// TwinCAT 3 PLC project state_machine_prj
// ProgramVersion: 3.1.4024.0
// libraries:
//   Tc2_Standard, * (Beckhoff Automation GmbH)
//   Tc2_System, * (Beckhoff Automation GmbH)
//   Tc2_Utilities, * (Beckhoff Automation GmbH)
//   Tc3_Module, * (Beckhoff Automation GmbH)
//   VisuDialogs, * (System)
// project tree:
//   DUTs/ ST_MyData.TcDUT
//   / GlobalTextList.TcGTLO, PlcTask.TcTTO, Visualization Manager.TcVMO (not stored)
//   POUs/ Class Diagram.TcCD (not stored), FB_ChargedState.TcPOU, FB_DischargeState.TcPOU, FB_DisconnectedState.TcPOU, FB_ErrorState.TcPOU, FB_FileWriter.TcPOU, FB_IdleState.TcPOU, FB_MACHINE.TcPOU, FB_PrechargeState.TcPOU, I_State.TcIO, MAIN.TcPOU
//   VISUs/ Visualisation.TcVIS
// (motion and I/O tree: see PLC project safety)
// real-time tasks:
//   TASK Safety: cycle T#5ms, priority 6, ADS port 350
//   TASK StateMachine: cycle T#1ms, priority 4, ADS port 351
// variable links:
//   safety/safety Instance <-> state_machine_prj/state_machine_prj Instance
//     PlcTask Outputs/MAIN.b_ESTOPout <-> PlcTask Inputs/MAIN.b_estop
//     PlcTask Outputs/MAIN.b_LED <-> PlcTask Inputs/MAIN.b_resetLed
//     PlcTask Outputs/MAIN.b_SafetyStateOut <-> PlcTask Inputs/MAIN.b_reset
//   state_machine_prj/state_machine_prj Instance <-> Device 5 (EtherCAT)/Term 1 (EK1100)/Term 2 (EL3702)
//     PlcTask Inputs/MAIN.n_A_sensors[0] <-> Ch2 Sample 0/Ch2 Value
//     PlcTask Inputs/MAIN.n_A_sensors[1] <-> Ch1 Sample 0/Ch1 Value
//   state_machine_prj/state_machine_prj Instance <-> Device 5 (EtherCAT)/Term 1 (EK1100)/Term 4 (EL3702)
//     PlcTask Inputs/MAIN.n_V_sensors[0] <-> Ch1 Sample 0/Ch1 Value
//     PlcTask Inputs/MAIN.n_V_sensors[1] <-> Ch2 Sample 0/Ch2 Value
//   state_machine_prj/state_machine_prj Instance <-> Device 5 (EtherCAT)/Term 1 (EK1100)/Term 6 (EL1004)
//     PlcTask Inputs/MAIN.b_bypass_contactors_fb[0] <-> Channel 3/Input
//     PlcTask Inputs/MAIN.b_bypass_contactors_fb[1] <-> Channel 4/Input
//     PlcTask Inputs/MAIN.b_main_contactors_fb[0] <-> Channel 1/Input
//     PlcTask Inputs/MAIN.b_main_contactors_fb[1] <-> Channel 2/Input
//   state_machine_prj/state_machine_prj Instance <-> Device 5 (EtherCAT)/Term 1 (EK1100)/Term 7 (EL2004)
//     PlcTask Outputs/MAIN.b_bypass_contactors[0] <-> Channel 3/Output
//     PlcTask Outputs/MAIN.b_bypass_contactors[1] <-> Channel 4/Output
//     PlcTask Outputs/MAIN.b_main_contactors[0] <-> Channel 1/Output
//     PlcTask Outputs/MAIN.b_main_contactors[1] <-> Channel 2/Output

CONFIGURATION state_machine_prj
    RESOURCE PLC ON TwinCAT3
        TASK PlcTask(INTERVAL := T#1ms, PRIORITY := 4);
        PROGRAM MAIN WITH PlcTask : MAIN;
    END_RESOURCE
END_CONFIGURATION

// ---- DUTs/ST_MyData.TcDUT
TYPE ST_MyData :
STRUCT
    Id          : UDINT;
    Value       : REAL;
    Timestamp   : T_MaxString; 
END_STRUCT
END_TYPE

// ---- POUs/I_State.TcIO
INTERFACE I_State

METHOD PUBLIC Check
END_METHOD

PROPERTY PUBLIC Description : STRING
GET
END_GET
END_PROPERTY

METHOD PUBLIC PressButton
END_METHOD

METHOD PUBLIC PressDischarge
END_METHOD

METHOD PUBLIC Reset
END_METHOD

METHOD PUBLIC Stop
END_METHOD

METHOD PUBLIC TimerDone
END_METHOD

END_INTERFACE

// ---- POUs/MAIN.TcPOU
PROGRAM MAIN
// Variables, constants ... are created (instanced) here
VAR
	(* Inputs *)
	n_V_sensors 				AT %I* 		: ARRAY[0..1] OF INT; // defining 2 elements array of INT type as input to the PLC task
	n_A_sensors 				AT %I*		: ARRAY[0..1] OF INT; 
	
	b_reset						AT %I*		: BOOL;
	b_estop						AT %I*		: BOOL;

	b_main_contactors_fb 		AT %I* 		: ARRAY[0..1] OF BOOL; // defining 4 elements array of BOOL type as input of feedback for the contactors to the PLC task
	b_bypass_contactors_fb 		AT %I* 		: ARRAY[0..1] OF BOOL;
	
	b_resetLed					AT %I*		: BOOL; 
	
	(* Outputs *)
	b_main_contactors			AT %Q*		: ARRAY[0..1] OF BOOL; // defining 4 elements array of BOOL type as outpout to the PLC task
	b_bypass_contactors			AT %Q*		: ARRAY[0..1] OF BOOL;

	(* FB_MACHINE *) 
	b_user_button							: BOOL := FALSE;
	b_discharge								: BOOL := FALSE;
	n_lower_boundV							: INT := 380;
	n_upper_boundV							: INT := 460; 
	n_minV 									: INT := 5;
	
	t_max_time								: TIME := T#250MS; //5x the time constant for a RC circuit with R=100ohms and C=235µF
	
	fbMachine 								: FB_MACHINE(nLowerBoundV := n_lower_boundV,
													     nUpperBoundV := n_upper_boundV,
													     nMinV := n_minV,
													     tMaxTime := t_max_time); 
	(*Visualisation variables*)
    sState         							: STRING;
	n_V_sensors_scaled 						: ARRAY[0..1] OF REAL; // defining 2 elements array of INT type as input to the PLC task
	n_A_sensors_scaled						: ARRAY[0..1] OF REAL;
	sLog									: ARRAY[0..19] OF STRING(600); 
	
	(* FILE_WRITER VARIABLES *) 
	sFilePath 								: STRING := 'C:\Users\Administrator\Desktop\AXav-Precharge_Curbs\'; //default file path for the data
    
	arrVoltageData    						: ARRAY [0..1] OF ST_MyData;
	arrCurrentData							: ARRAY [0..1] OF ST_MyData;
	arrBypassData							: ARRAY [0..1] OF ST_MyData;
	arrMainData								: ARRAY [0..1] OF ST_MyData;
	
    nIteration      						: UDINT:=0;
    bStartNewJob    						: BOOL := FALSE; // When set to false the FileWriter is active
	bFirstLoop								: BOOL := TRUE; // Allows to write the header of the file on the first loop (then it will be set to FALSE for the rest of the task)
	tStartTime								: TIME;
	
	fbVoltage1								: FB_FileWriter; 
	fbCurrent1								: FB_FileWriter; 
	fbVoltage2								: FB_FileWriter;
	fbCurrent2								: FB_FileWriter;
	fbBypass1								: FB_FileWriter;
	fbBypass2								: FB_FileWriter; 
	fbMain1									: FB_FileWriter; 
	fbMain2									: FB_FileWriter; 
	
	fbFormatString  						: FB_FormatString;
	fbFormatString1  						: FB_FormatString;
	fbFormatString2							: FB_FormatString; 
	fbFormatString3							: FB_FormatString;
	
	sHeader									: STRING := 'ID;VALUE;TIMESTAMP$n';

	n_Idx									: INT := 0;
	fileBlocks 								: ARRAY[0..3] OF  FB_FileWriter := [fbCurrent1, fbCurrent2, fbVoltage1, fbVoltage2];
	fileBlocksContactors					: ARRAY[0..3] OF  FB_FileWriter := [fbBypass1, fbBypass2, fbMain1, fbMain2];
    s_fileNames 							: ARRAY[0..3] OF STRING := ['SupplyCurrent.txt', 'LoadCurrent.txt', 'SupplyVoltage.txt', 'LoadVoltage.txt'];
	s_fileNamesContactors					: ARRAY[0..3] OF STRING := ['BypassContactor1.txt', 'BypassContactor2.txt', 'MainContactor1.txt', 'MainContactor2.txt'];
	s_FBStates								: ARRAY[0..3] OF STRING;
	s_FBStatesContactors					: ARRAY[0..3] OF STRING; 
END_VAR

(* ---------------------------- STATE MACHINE ------------------------------- *) 
fbMachine.Run(
			bAck:=b_user_button, 
			bDischarge := b_discharge, 
			nVSensors := n_V_Sensors, 
			nASensors := n_A_Sensors, 
			bBypassContactorsFB := b_bypass_contactors_fb,
			bMainContactorsFB := b_main_contactors_fb,
			bReset := b_reset,
			bESTOP := b_estop,
			bMainContactors => b_main_contactors, 
			bBypassContactors => b_bypass_contactors,
			);

(* --------------------- Visualisation properties ---------------------- *) 
// I need to link local variables with "fbMachine" properties because it is not possible to link a visualisation object (e.g. textbox) with a function box property
sState := fbMachine.ipState.Description;
n_V_sensors_scaled := fbMachine.VSensors; 
n_A_sensors_scaled := fbMachine.ASensors; 
sLog := fbMachine.Logs; 

(* --------------------- Data Saving ----------------------------- *)	
FOR n_Idx := 0 TO 3 DO
	fileBlocks[n_Idx](
		sFileName := s_fileNames[n_Idx],
		sFilePath := sFilePath,
		sNetId    := '');
		
	fileBlocksContactors[n_Idx](
		sFileName := s_fileNamesContactors[n_Idx],
		sFilePath := sFilePath,
		sNetId    := '');
			
	s_FBStates[n_Idx] := fileBlocks[n_Idx].FileWriteState; // STRING states to display in the visualisation file
	s_FBStatesContactors[n_Idx] := fileBlocksContactors[n_Idx].FileWriteState; // STRING states to display in the visualisation file
END_FOR	

IF bFirstLoop THEN // On the first loop
	FOR n_Idx := 0 TO 3 DO
		fileBlocks[n_Idx].WriteToFile(message := sHeader); // write the header of the file 
		fileBlocksContactors[n_Idx].WriteToFile(message := sHeader); // write the header of the file 
	END_FOR	
	tStartTime := TIME();
	bFirstLoop := FALSE;
END_IF

IF bStartNewJob THEN 
	// save the new data to the struct variable
	FOR n_Idx := 0 TO 1 DO
		arrVoltageData[n_Idx].Id := nIteration;
		arrVoltageData[n_Idx].Value := n_V_sensors_scaled[n_Idx];
		arrVoltageData[n_Idx].Timestamp := DINT_TO_STRING(TO_DINT(TIME() - tStartTime));
	
		arrCurrentData[n_Idx].Id := nIteration;
		arrCurrentData[n_Idx].Value :=n_A_sensors_scaled[n_Idx];
		arrCurrentData[n_Idx].Timestamp := DINT_TO_STRING(TO_DINT(TIME() - tStartTime)); 
		
		arrBypassData[n_Idx].Id := nIteration;
		arrBypassData[n_Idx].Value := BOOL_TO_REAL(b_bypass_contactors_fb[n_Idx]);
		arrBypassData[n_Idx].Timestamp := DINT_TO_STRING(TO_DINT(TIME() - tStartTime));
	
		arrMainData[n_Idx].Id := nIteration;
		arrMainData[n_Idx].Value :=BOOL_TO_REAL(b_main_contactors[n_Idx]);
		arrMainData[n_Idx].Timestamp := DINT_TO_STRING(TO_DINT(TIME() - tStartTime)); 
	END_FOR
	// write the data in the text file 
	FOR n_Idx := 0 TO 1 DO
		fbFormatString(
			sFormat := '%d;%f;%s$n',
			arg1    := F_UDINT(arrCurrentData[n_Idx].Id),
			arg2    := F_REAL(arrCurrentData[n_Idx].Value),
			arg3    := F_STRING(arrCurrentData[n_Idx].Timestamp));
		fileBlocks[n_Idx].WriteToFile(fbFormatString.sOut);
		fbFormatString1(
			sFormat := '%d;%f;%s$n',
			arg1    := F_UDINT(arrVoltageData[n_Idx].Id),
			arg2    := F_REAL(arrVoltageData[n_Idx].Value),
			arg3    := F_STRING(arrVoltageData[n_Idx].Timestamp));
		fileBlocks[n_Idx+2].WriteToFile(fbFormatString1.sOut);
		fbFormatString2(
			sFormat := '%d;%f;%s$n',
			arg1    := F_UDINT(arrBypassData[n_Idx].Id),
			arg2    := F_REAL(arrBypassData[n_Idx].Value),
			arg3    := F_STRING(arrBypassData[n_Idx].Timestamp));
		fileBlocksContactors[n_Idx].WriteToFile(fbFormatString2.sOut);
		fbFormatString3(
			sFormat := '%d;%f;%s$n',
			arg1    := F_UDINT(arrMainData[n_Idx].Id),
			arg2    := F_REAL(arrMainData[n_Idx].Value),
			arg3    := F_STRING(arrMainData[n_Idx].Timestamp));
		fileBlocksContactors[n_Idx+2].WriteToFile(fbFormatString3.sOut);
	END_FOR
	nIteration := nIteration + 1;
END_IF

END_PROGRAM

// ---- POUs/FB_MACHINE.TcPOU
FUNCTION_BLOCK PUBLIC FB_MACHINE

VAR_INPUT
	nVSensors 		 				: ARRAY[0..1] OF INT; // 2 INT elements array which contains the voltage sensors outputs
	nASensors 						: ARRAY[0..1] OF INT; // 2 INT elements array whihch contains the current sensors outputs
	
	(* Pre-Charge Timer *) 
	tMaxTime						: TIME; // Maximum pre-charge time
	
	(* Voltage boundaries *) 
	nLowerBoundV					: INT; // Input voltage lower bound (~50V) 
	nUpperBoundV					: INT; // Input voltage upper bound (~200V)
	nMinV							: INT; // Minimum voltage to leave "disconnected" state
	
	(* Timer *)
	charge_TON						: TON; 
END_VAR

VAR_OUTPUT
	ipState 						: I_State := fbDisconnectedState; // Current State of the state machine (default is FB_DisconnectedState)
END_VAR

VAR (* Internal variables *)
	fbDisconnectedState 			: FB_DisconnectedState(THIS);	
	fbIdleState 					: FB_IdleState(THIS); 
	fbPrechargeState 				: FB_PrechargeState(THIS); 
	fbChargedState					: FB_ChargedState(THIS); 
	fbDischargeState				: FB_DischargeState(THIS);
	fbErrorState					: FB_ErrorState(THIS);
	
	(* Sensors scaling *) 
	n_idx_1 						: INT := 0; 
	fVSensorsScaled 				: ARRAY[0..1] OF REAL; // defining 2 elements array of REAL type as internal variables
	fASensorsScaled 				: ARRAY[0..1] OF REAL; 
	
	(* Message log *) 
	sLog 							: ARRAY [0..19] OF STRING(600);
	nCount							: UINT := 0; // Keeps track of the number of elements in the array	
	nArraySize 						: UINT := 20; // Edit value if size of sLog changes 
	tLaunchTime 					: TIME; 	
	sMessage						: STRING(600);
	sPrevMessage					: STRING(600);
	
	(* Contactors *)
	bMainContactors					: ARRAY[0..1] OF BOOL; 
	bBypassContactors 				: ARRAY[0..1] OF BOOL; 
	
	(* Contactors feedback *)
	bMainContactorsFB				: ARRAY[0..1] OF BOOL; // defining 2 elements array of BOOL type as input of feedback for the main contactors to the PLC task
	bBypassContactorsFB				: ARRAY[0..1] OF BOOL; // defining 2 elements array of BOOL type as input of feedback for the precharge contactors to the PLC task

	(* Triggers *) 
	rtrigButtonAck					: R_TRIG; // Define trigger for user button 
	rtrigButtonDisch				: R_TRIG; 
	
	(* Misc *) 
	nRunCounter						: UINT := 10;
END_VAR

tLaunchTime := TIME(); // Reference point for log messages

METHOD PRIVATE AddToLog
VAR_INPUT
	sMsgINPUT			: STRING(600); //different from Message that doesn't contain the time tag
END_VAR
VAR
	nIdx 				: UINT := 0;
END_VAR
// IF the ARRAY is full, remove the first element 
IF NOT(Message = PrevMessage) THEN // NOT sMsgINPUT BECAUSE IT CONTAINS THE TIME TAG which will make it always different from PrevMessage
	IF THIS^.nCount = THIS^.nArraySize THEN
		FOR nIdx := 0 TO THIS^.nArraySize - 2 DO 
			sLog[nIdx] := sLog[nIdx + 1 ]; // shift the whole array
		END_FOR
		sLog[THIS^.nCount - 1] := sMsgINPUT; // Add the new string as the last elemnt of the array
	ELSE
		sLog[THIS^.nCount] := sMsgINPUT;
		THIS^.nCount := THIS^.nCount + 1;
	END_IF 
	THIS^.PrevMessage := Message;
END_IF
END_METHOD

PROPERTY PUBLIC ASensors : ARRAY[0..1] OF REAL
GET
ASensors := THIS^.fASensorsScaled;
END_GET
END_PROPERTY

PROPERTY PUBLIC BypassContactors : ARRAY[0..1] OF BOOL
GET
BypassContactors := THIS^.bBypassContactors;
END_GET
SET
THIS^.bBypassContactors := BypassContactors;
END_SET
END_PROPERTY

PROPERTY PRIVATE BypassContactorsFB : ARRAY[0..1] OF BOOL
GET
BypassContactorsFB := THIS^.bBypassContactorsFB;
END_GET
SET
THIS^.bBypassContactorsFB := BypassContactorsFB;
END_SET
END_PROPERTY

PROPERTY PUBLIC ChargedState : I_State
GET
ChargedState := THIS^.fbChargedState;
END_GET
END_PROPERTY

METHOD CheckContactors
VAR
	nIdx							: INT := 0; 
	
	bMainContactorsCheck 			: BOOL := TRUE; // true means that there is no problem
	bBypassContactorsCheck 			: BOOL := TRUE; 
	bConclusion 					: BOOL := TRUE; // true means that there is no problem
	
	fbDischargeState				: FB_DischargeState(THIS);
END_VAR
FOR nIdx := 0 TO 1 DO 
	bMainContactorsCheck := THIS^.bMainContactors[nIdx] = THIS^.bMainContactorsFB[nIdx]; // checks that the feedback signal corresponds to the contactor state
	bBypassContactorsCheck := THIS^.bBypassContactors[nIdx] = THIS^.bBypassContactorsFB[nIdx];
	
	IF NOT(bMainContactorsCheck) THEN
		THIS^.Message := CONCAT('[CheckContactors] The ', CONCAT(INT_TO_STRING(nIdx), ' Main contactor state does not match the signal sent'));
		bConclusion := FALSE; 
	END_IF
	IF NOT(bBypassContactorsCheck) THEN
		THIS^.Message := CONCAT('[CheckContactors] The ', CONCAT(INT_TO_STRING(nIdx), ' Bypass contactor state does not match the signal sent'));
		bConclusion := FALSE; 
	END_IF
END_FOR 

IF NOT(bConclusion) THEN
	THIS^.Message := CONCAT(THIS^.Message, '[CheckContactors]$A0 THE SYSTEM IS NOW BEING DISHCARGED');  
	THIS^.SetState(fbDischargeState);
	bConclusion := TRUE;
END_IF
END_METHOD

PROPERTY PUBLIC DischargeState : I_State
GET
DischargeState :=  THIS^.fbDischargeState;
END_GET
END_PROPERTY

PROPERTY PUBLIC DisconnectedState : I_State
GET
DisconnectedState := THIS^.fbDisconnectedState;
END_GET
END_PROPERTY

PROPERTY PUBLIC ErrorState : I_State
GET
ErrorState := THIS^.fbErrorState;
END_GET
END_PROPERTY

METHOD FB_init 
VAR_INPUT
	bInitRetains : BOOL; // if TRUE, the retain variables are initialized (warm start / cold start)
	bInCopyCode : BOOL;  // if TRUE, the instance afterwards gets moved into the copy code (online change)
	
	(* Pre-Charge Timer *) 
	tMaxTime						: TIME; 
	
	(* Voltage boundaries *) 
	nLowerBoundV					: INT; // Input voltage lower bound (~50V) 
	nUpperBoundV					: INT; // Input voltage upper bound (~200V)
	nMinV							: INT; // Minimum voltage to leave "disconnected" state
END_VAR
THIS^.tMaxTime := tMaxTime;
THIS^.nLowerBoundV := nLowerBoundV; 
THIS^.nUpperBoundV := nUpperBoundV; 
THIS^.nMinV := nMinV;
END_METHOD

PROPERTY PUBLIC IdleState : I_State
GET
IdleState := THIS^.fbIdleState;
END_GET
END_PROPERTY

PROPERTY PUBLIC Logs : ARRAY[0..19] OF STRING(600)
GET
Logs := THIS^.sLog;
END_GET
END_PROPERTY

PROPERTY PUBLIC LowerBoundV : INT
GET
LowerBoundV := THIS^.nLowerBoundV;
END_GET
SET
THIS^.nLowerBoundV := LowerBoundV;
END_SET
END_PROPERTY

PROPERTY PUBLIC MainContactors : ARRAY[0..1] OF BOOL
GET
MainContactors := THIS^.bMainContactors;
END_GET
SET
THIS^.bMainContactors := MainContactors;
END_SET
END_PROPERTY

PROPERTY PRIVATE MainContactorsFB : ARRAY[0..1] OF BOOL
GET
MainContactorsFB := THIS^.bMainContactorsFB;
END_GET
SET
THIS^.bMainContactorsFB := MainContactorsFB;
END_SET
END_PROPERTY

PROPERTY PUBLIC Message : STRING(600)
GET // PUBLIC
Message := THIS^.sMessage;
END_GET
SET // PUBLIC
THIS^.sMessage := Message; 
// Adds the difference between the laucnh time and the current time at the beginning of the log message
THIS^.AddToLog(CONCAT(CONCAT(CONCAT('[', TIME_TO_STRING(TIME()-THIS^.tLaunchTime)), '] '), THIS^.sMessage));
END_SET
END_PROPERTY

PROPERTY PUBLIC MinV : INT
GET
MinV := THIS^.nMinV;
END_GET
SET
THIS^.nMinV := MinV;
END_SET
END_PROPERTY

PROPERTY PUBLIC PrechargeState : I_State
GET
PrechargeState := THIS^.fbPrechargeState;
END_GET
END_PROPERTY

PROPERTY PrevMessage : STRING(600)
GET
PrevMessage := THIS^.sPrevMessage;
END_GET
SET
THIS^.sPrevMessage := PrevMessage;
END_SET
END_PROPERTY

METHOD PUBLIC Run
VAR_INPUT
	(* User buttons *)
	bAck							: BOOL; // User "next state" button
	bDischarge						: BOOL; // User "discharge" trigger button
	
	(* Sensors *)
	nVSensors 		 				: ARRAY[0..1] OF INT; // defining 2 elements array of INT type as input to the PLC task
	nASensors 						: ARRAY[0..1] OF INT; 
	
	bMainContactorsFB				: ARRAY[0..1] OF BOOL; 
	bBypassContactorsFB				: ARRAY[0..1] OF BOOL;
	
	bReset							: BOOL; // Reset signal
	bESTOP							: BOOL; // TRUE when the button is pressed
END_VAR

VAR
END_VAR

VAR_OUTPUT
	bMainContactors					: ARRAY[0..1] OF BOOL; 
	bBypassContactors				: ARRAY[0..1] OF BOOL;
END_VAR
(* ------------------------------------- SAFETY ------------------------------------ *)
//E-Stop check
IF NOT(bESTOP) THEN	
	ipState.Stop(); // sets state to ErrorState
	ipState.Check(); 
	bMainContactors := THIS^.MainContactors; 
	bBypassContactors := THIS^.BypassContactors;
	RETURN;
END_IF
//Reset check
IF ipState = ErrorState AND bReset THEN // reset has been pressed 
	ipState.Reset();
END_IF
// Functionning contactors check
IF RunCounter MOD 15 = 0  THEN // Checks contactors every 15 run loop because it takes some time for the feedback to adjust
	CheckContactors(); // Ensures that the contactors signals are the same as the contactors states
END_IF


(* ---------------------------------- STATE MACHINE ------------------------------------ *) 

(*Contactors*)
THIS^.MainContactorsFB := bMainContactorsFB;
THIS^.BypassContactorsFB := bBypassContactorsFB;

(* Buttons*) 
rtrigButtonAck(CLK := bAck); // Sets trigger for bUserButton variable 
rtrigButtonDisch(CLK := bDischarge); 

(*Sensors*)
THIS^.nVSensors := nVSensors;
THIS^.nASensors := nASensors; 

(* Timer configuration *) 
charge_TON(PT := THIS^.tMaxTime);

THIS^.ScaleSensors(); // Scaling the values of the sensors which will be used in the state machine 

IF (charge_TON.Q) THEN
	ipState.TimerDone(); // Used for the precharge state 
END_IF

IF (rtrigButtonDisch.Q) THEN
	ipState.PressDischarge();
END_IF

IF (rtrigButtonAck.Q) THEN
	ipState.PressButton();
END_IF

ipState.Check(); 

// Output of the state machine
bMainContactors := THIS^.MainContactors; 
bBypassContactors := THIS^.BypassContactors;
RETURN;
END_METHOD

PROPERTY PRIVATE RunCounter : UINT
GET
RunCounter := THIS^.nRunCounter;
END_GET
SET
THIS^.nRunCounter := RunCounter;
END_SET
END_PROPERTY

METHOD PRIVATE ScaleSensors
// Scaling of V sensors
FOR n_idx_1 := 0 TO 1 DO
	fVSensorsScaled[n_idx_1] := 1000*INT_TO_REAL(THIS^.nVSensors[n_idx_1])/32768;
	// e.g., if 1000 V on sensor --> card measures +10V --> software value = 32767 --> scaling is therefore 1000*VAL/32768
END_FOR

FOR n_idx_1 := 0 TO 1 DO
	fASensorsScaled[n_idx_1] := 25*INT_TO_REAL(THIS^.nASensors[n_idx_1])/32768; 
END_FOR
END_METHOD

METHOD INTERNAL SetState
VAR_INPUT
	newState		: I_State;
END_VAR
THIS^.ipState := newState;
END_METHOD

PROPERTY PUBLIC UpperBoundV : INT
GET
UpperBoundV := THIS^.nUpperBoundV;
END_GET
SET
THIS^.nUpperBoundV := UpperBoundV;
END_SET
END_PROPERTY

PROPERTY PUBLIC VSensors : ARRAY[0..1] OF REAL
GET
VSensors := THIS^.fVSensorsScaled;
END_GET
END_PROPERTY

END_FUNCTION_BLOCK

// ---- POUs/FB_DisconnectedState.TcPOU
FUNCTION_BLOCK INTERNAL FB_DisconnectedState IMPLEMENTS I_State
VAR
	pMachine		: POINTER TO FB_Machine; // Points to the state machine (THIS)
	fVSensors		: ARRAY[0..1] OF REAL; 
END_VAR

METHOD PUBLIC Check
VAR
	fInputVoltage 		: REAL; 
END_VAR
THIS^.ResetContactors(); //THE CONTACTORS NEED TO ALWAYS BE OPEN IN THIS STATE
fVSensors := THIS^.pMachine^.VSensors;
fInputVoltage := fVSensors[0];

IF (fInputVoltage >= THIS^.pMachine^.MinV) THEN
	THIS^.pMachine^.Message := '[DISCONNECTED] The input voltage is >= than the minimum voltage. $0A WAITING FOR ACKNOWLEDGEMENT TO ENTER IDLE STATE;';
ELSE 
	THIS^.pMachine^.Message := '[DISCONNECTED]The input voltage is <= than the minimum voltage.';
END_IF
END_METHOD

PROPERTY PUBLIC Description : STRING
GET
Description := 'DISCONNECTED';
END_GET
END_PROPERTY

METHOD PUBLIC FB_init
VAR_INPUT
	bInitRetains 	: BOOL; // if TRUE, the retain variables are initialized (warm start / cold start)
	bInCopyCode 	: BOOL;  // if TRUE, the instance afterwards gets moved into the copy code (online change)
	pMachine		: POINTER TO FB_Machine; // Points to the state machine (THIS)
END_VAR
THIS^.pMachine := pMachine;
END_METHOD

METHOD PUBLIC PressButton 
VAR
	//fbIdleSTate		: FB_IdleState(THIS^.pMachine); => variable for changing state method that causes a PLC bug
	fInputVoltage		: REAL; 
END_VAR
fVSensors := THIS^.pMachine^.VSensors;
fInputVoltage := fVSensors[0];

IF (fInputVoltage >= THIS^.pMachine^.MinV) THEN
		//THIS^.pMachine^.SetState(fbIdleState); => changing state method that causes a PLC bug
		THIS^.pMachine^.Message := '[DISCONNECTED] Acknowledge button has been pressed. $0A SYSTEM ENTERS IDLE STATE.';
		THIS^.pMachine^.SetState(THIS^.pMachine^.IdleState);
END_IF
END_METHOD

METHOD PUBLIC PressDischarge
END_METHOD

METHOD PUBLIC Reset
END_METHOD

METHOD PUBLIC ResetContactors
VAR
	nIdx					: INT := 0; 
	bBypassContactors		: ARRAY[0..1] OF BOOL; 
	bMainContactors			: ARRAY[0..1] OF BOOL; 
END_VAR
FOR nIdx := 0 TO 1 BY 1 DO 
	bBypassContactors[nIdx] := FALSE;
	bMainContactors[nIdx] := FALSE; 
END_FOR

THIS^.pMachine^.BypassContactors := bBypassContactors; // Reset every contactor 
THIS^.pMachine^.MainContactors := bMainContactors;
END_METHOD

METHOD PUBLIC Stop
THIS^.pMachine^.SetState(THIS^.pMachine^.ErrorState);
END_METHOD

METHOD PUBLIC TimerDone
END_METHOD

END_FUNCTION_BLOCK

// ---- POUs/FB_IdleState.TcPOU
FUNCTION_BLOCK INTERNAL FB_IdleState IMPLEMENTS I_State
VAR
	pMachine				: POINTER TO FB_Machine; // Points to the state machine (THIS)
	fVSensors				: ARRAY [0..1] OF REAL; 
END_VAR

METHOD PUBLIC Check 
VAR
	fInputVoltage			: REAL;	
END_VAR
fVSensors := THIS^.pMachine^.VSensors;

fInputVoltage := fVSensors[0];

IF (fInputVoltage >= THIS^.pMachine^.LowerBoundV AND fInputVoltage <= THIS^.pMachine^.UpperBoundV) THEN
	THIS^.pMachine^.Message := '[IDLE]The input voltage is within the boundaries.$0A NOW WAITING FOR ACKNOWLEDGEMENT TO ENTER PRE-CHARGE STATE.';
ELSE
	THIS^.pMachine^.Message := '[IDLE] The input voltage is NOT within the boundaries.$0A SYSTEM ENTERS DISCHARGE STATE.';
	THIS^.pMachine^.SetState(THIS^.pMachine^.DischargeState);
END_IF
END_METHOD

PROPERTY PUBLIC Description : STRING
GET
Description := 'IDLE';
END_GET
END_PROPERTY

METHOD PUBLIC FB_init
VAR_INPUT
	bInitRetains 	: BOOL; // if TRUE, the retain variables are initialized (warm start / cold start)
	bInCopyCode 	: BOOL;  // if TRUE, the instance afterwards gets moved into the copy code (online change)
	pMachine		: POINTER TO FB_Machine; // Points to the state machine (THIS)
END_VAR
THIS^.pMachine := pMachine;
END_METHOD

METHOD PUBLIC PressButton
VAR
	fInputVoltage			: REAL; 
END_VAR
fVSensors := THIS^.pMachine^.VSensors;
fInputVoltage := fVSensors[0];

IF (fInputVoltage >= THIS^.pMachine^.LowerBoundV AND fInputVoltage <= THIS^.pMachine^.UpperBoundV) THEN
	THIS^.pMachine^.Message := '[IDLE] Acknowledge button has been pressed. $0A SYSTEM ENTERS PRECHARGE STATE.';
	THIS^.pMachine^.SetState(THIS^.pMachine^.PrechargeState);
	THIS^.StartTimer();
END_IF
END_METHOD

METHOD PUBLIC PressDischarge
THIS^.pMachine^.Message := '[IDLE] Discharge button has been pressed. $0A SYSTEM ENTERS DISCHARGE STATE.';
THIS^.pMachine^.SetState(THIS^.pMachine^.DischargeState);
END_METHOD

METHOD PUBLIC Reset
THIS^.pMachine^.Message := '[IDLE] Reset button has been pressed. $0A SYSTEM ENTERS DISCHARGE STATE.';
THIS^.pMachine^.SetState(THIS^.pMachine^.DischargeState);
END_METHOD

METHOD PUBLIC StartTimer
THIS^.pMachine^.charge_TON.IN := TRUE; // Starts the Timer
END_METHOD

METHOD PUBLIC Stop
THIS^.pMachine^.SetState(THIS^.pMachine^.ErrorState);
END_METHOD

METHOD PUBLIC TimerDone
END_METHOD

END_FUNCTION_BLOCK

// ---- POUs/FB_PrechargeState.TcPOU
FUNCTION_BLOCK INTERNAL FB_PrechargeState  IMPLEMENTS I_State
VAR
	pMachine				: POINTER TO FB_Machine; // Points to the state machine (THIS)
	fVSensors				: ARRAY [0..1] OF REAL;
END_VAR

METHOD PUBLIC Check
VAR
	fLoadVoltage			: REAL;
	fInputVoltage 			: REAL;
END_VAR
THIS^.SetMainContactors();
fVSensors := THIS^.pMachine^.VSensors;

fInputVoltage := fVSensors[0];
fLoadVoltage := fVSensors[1];

IF (fLoadVoltage > 1.1 * fInputVoltage) THEN
	(* If the load voltage is greater than 110% of the input voltage then we consider that there is a problem and the load is disconnected *)
	THIS^.pMachine^.Message := '[PRECHARGE] The load voltage is greater than 110 percent of the input voltage.$0A THE SYSTEM ENTERS DISCHARGE STATE';
	THIS^.pMachine^.SetState(THIS^.pMachine^.DischargeState); 
	
ELSIF (fLoadVoltage <= 1.1 * fInputVoltage AND fLoadVoltage >= 0.9502 * fInputVoltage) THEN
	THIS^.ResetTimer();
	THIS^.pMachine^.Message := '[PRECHARGE]The load voltage is within the boundaries.$0A WAITING FOR USER ACKNOWLEDGMENT TO ENTER CHARGE STATE.';
END_IF;
END_METHOD

PROPERTY PUBLIC Description : STRING
GET
Description := 'PRE-CHARGE';
END_GET
END_PROPERTY

METHOD PUBLIC FB_init
VAR_INPUT
	bInitRetains : BOOL; // if TRUE, the retain variables are initialized (warm start / cold start)
	bInCopyCode : BOOL;  // if TRUE, the instance afterwards gets moved into the copy code (online change)
	pMachine		: POINTER TO FB_Machine; // Points to the state machine (THIS)
END_VAR
THIS^.pMachine := pMachine;
END_METHOD

METHOD PUBLIC PressButton
VAR
	fLoadVoltage			: REAL;
	fInputVoltage 			: REAL;
END_VAR
fVSensors := THIS^.pMachine^.VSensors;
fInputVoltage := fVSensors[0];
fLoadVoltage := fVSensors[1];

IF (fLoadVoltage <= 1.1 * fInputVoltage AND fLoadVoltage >= 0.9502 * fInputVoltage) THEN
	THIS^.ResetTimer(); // Not necessary, here for redundancy 
	THIS^.pMachine^.SetState(THIS^.pMachine^.ChargedState);	
	THIS^.pMachine^.Message := '[PRECHARGE] Acknowledge button has been pressed. $0A SYSTEM ENTERS CHARGED STATE.';
END_IF
END_METHOD

METHOD PUBLIC PressDischarge
THIS^.pMachine^.Message := '[PRECHARGE] Discharge button has been pressed. $0A SYSTEM ENTERS DISCHARGE STATE.';
THIS^.pMachine^.SetState(THIS^.pMachine^.DischargeState);
END_METHOD

METHOD PUBLIC Reset
THIS^.pMachine^.Message := '[PRECHARGE] Reset button has been pressed. $0A SYSTEM ENTERS DISCHARGE STATE.';
THIS^.pMachine^.SetState(THIS^.pMachine^.DischargeState);
END_METHOD

METHOD PUBLIC ResetMainContactors
VAR
	nIdx				: INT;
	bMainContactors		: ARRAY[0..1] OF BOOL;
END_VAR
FOR nIdx := 0 TO 1 DO
	bMainContactors[nIdx] := FALSE; 
END_FOR

THIS^.pMachine^.MainContactors := bMainContactors;
END_METHOD

METHOD PUBLIC ResetTimer
THIS^.pMachine^.charge_TON.IN := FALSE;
END_METHOD

METHOD PUBLIC SetMainContactors
VAR
	nIdx				: INT;
	bMainContactors		: ARRAY[0..1] OF BOOL;
END_VAR
FOR nIdx := 0 TO 1 DO
	bMainContactors[nIdx] := TRUE; 
END_FOR

THIS^.pMachine^.MainContactors := bMainContactors;
END_METHOD

METHOD PUBLIC Stop
THIS^.pMachine^.SetState(THIS^.pMachine^.ErrorState);
END_METHOD

METHOD PUBLIC TimerDone
THIS^.pMachine^.Message := '[PRECHARGE] The charging time has exceeded the set limit.$0A THE SYSTEM ENTERS DISCHARGE STATE'; 		 

THIS^.ResetTimer(); 

THIS^.pMachine^.SetState(THIS^.pMachine^.DischargeState);
END_METHOD

END_FUNCTION_BLOCK

// ---- POUs/FB_ChargedState.TcPOU
FUNCTION_BLOCK INTERNAL FB_ChargedState IMPLEMENTS I_State
VAR
	pMachine				: POINTER TO FB_Machine; // Points to the state machine (THIS)	
	fVSensors 				: ARRAY[0..1] OF REAL;
END_VAR

METHOD PUBLIC Check 
VAR
	fInputVoltage			: REAL;
	fLoadVoltage 			: REAL; 
END_VAR
THIS^.SetMainContactors(); // not necessary but reinforces safety 
THIS^.SetBypassContactors(); // necessary

fVSensors := THIS^.pMachine^.VSensors;

fLoadVoltage := fVSensors[1];
fInputVoltage := fVSensors[0];

IF (fLoadVoltage <= 1.1 * fInputVoltage AND fLoadVoltage >= 0.9502 * fInputVoltage) THEN
	IF (fInputVoltage >= THIS^.pMachine^.LowerBoundV AND fInputVoltage <= THIS^.pMachine^.UpperBoundV) THEN
		THIS^.pMachine^.Message := '[CHARGED] The input and load voltages are within the boundaries. $0A PRESS "DISCHARGE" TO ENTER DISCHARGE STATE';
  	ELSE 
		THIS^.pMachine^.Message := '[CHARGED] The load voltage corresponds to the input voltage, but is not included within the defined limits.$0A THE SYSTEM ENTERS DISCHARGE STATE';
		THIS^.pMachine^.SetState(THIS^.pMachine^.DischargeState);
	END_IF
 
ELSE
	THIS^.pMachine^.Message := '[CHARGED] The load voltage DOES NOT match the input voltage.$0A THE SYSTEM ENTERS DISCHARGE STATE';
	THIS^.pMachine^.SetState(THIS^.pMachine^.DischargeState);
END_IF
END_METHOD

PROPERTY PUBLIC Description : STRING
GET
Description := 'CHARGED';
END_GET
END_PROPERTY

METHOD PUBLIC FB_init 
VAR_INPUT
	bInitRetains 	: BOOL; // if TRUE, the retain variables are initialized (warm start / cold start)
	bInCopyCode 	: BOOL;  // if TRUE, the instance afterwards gets moved into the copy code (online change)
	
	pMachine		: POINTER TO FB_Machine; // Points to the state machine (THIS)
END_VAR
THIS^.pMachine := pMachine;
END_METHOD

METHOD PUBLIC PressButton
END_METHOD

METHOD PUBLIC PressDischarge
THIS^.pMachine^.Message := '[CHARGED] Discharge button has been pressed. $0A SYSTEM ENTERS DISCHARGE STATE.';
THIS^.pMachine^.SetState(THIS^.pMachine^.DischargeState);
END_METHOD

METHOD PUBLIC Reset
THIS^.pMachine^.Message := '[CHARGED] Reset button has been pressed. $0A SYSTEM ENTERS DISCHARGE STATE.';
THIS^.pMachine^.SetState(THIS^.pMachine^.DischargeState);
END_METHOD

METHOD PUBLIC SetBypassContactors
VAR
	nIdx				: INT;
	bBypassContactors	: ARRAY[0..1] OF BOOL;
END_VAR
FOR nIdx := 0 TO 1 DO 
	bBypassContactors[nIdx] := TRUE; 
END_FOR

THIS^.pMachine^.BypassContactors := bBypassContactors;
END_METHOD

METHOD PUBLIC SetMainContactors
VAR
	nIdx				: INT;
	bMainContactors 	: ARRAY[0..1] OF BOOL;
END_VAR
FOR nIdx := 0 TO 1 DO 
	bMainContactors[nIdx] := TRUE;
END_FOR

THIS^.pMachine^.MainContactors := bMainContactors;
END_METHOD

METHOD PUBLIC Stop
THIS^.pMachine^.SetState(THIS^.pMachine^.ErrorState);
END_METHOD

METHOD PUBLIC TimerDone
END_METHOD

END_FUNCTION_BLOCK

// ---- POUs/FB_DischargeState.TcPOU
FUNCTION_BLOCK INTERNAL FB_DischargeState IMPLEMENTS I_State
VAR
	pMachine		: POINTER TO FB_Machine; // Points to the state machine (THIS)
	fVSensors		: ARRAY [0..1] OF REAL; 
END_VAR

METHOD PUBLIC Check
VAR
	fLoadVoltage			: REAL; 
	fInputVoltage			: REAL; 
END_VAR
THIS^.ResetContactors(); // THE CONTACTORS NEED TO ALAWAYS BE OPEN IN THIS STATE NO MATTER WHAT WAS THE PREVIOUS STATE
THIS^.ResetTimer(); // in case the emergency stop is pressed while the circuit is in precharge state
fVSensors := THIS^.pMachine^.VSensors;

fInputVoltage := fVSensors[0];
fLoadVoltage := fVSensors[1];

IF (fLoadVoltage < 0.1 * fInputVoltage) THEN
	THIS^.pMachine^.Message := '[DISCHARGE] The load voltage is now less than 1 percent of the input voltage.$0A WAITING FOR ACKNOWLEDGEMENT TO DISCONNECT SYSTEM.';
ELSE 
	THIS^.pMachine^.Message := '[DISCHARGE] Waiting for load voltage to be lower than 10 percent of the input voltage.';
END_IF
END_METHOD

PROPERTY PUBLIC Description : STRING
GET
Description := 'DISCHARGE';
END_GET
END_PROPERTY

METHOD PUBLIC FB_init
VAR_INPUT
	bInitRetains : BOOL; // if TRUE, the retain variables are initialized (warm start / cold start)
	bInCopyCode : BOOL;  // if TRUE, the instance afterwards gets moved into the copy code (online change)
	pMachine		: POINTER TO FB_Machine; // Points to the state machine (THIS)
END_VAR
THIS^.pMachine := pMachine;
END_METHOD

METHOD PUBLIC PressButton 
VAR
	fLoadVoltage		: REAL; 
	fInputVoltage		: REAL; 
END_VAR
fVSensors := THIS^.pMachine^.VSensors;
fInputVoltage := fVSensors[0];
fLoadVoltage := fVSensors[1];

IF (fLoadVoltage < 0.1 * fInputVoltage) THEN
	THIS^.pMachine^.Message := '[DISCHARGE] Acknowledge button has been pressed. $0A SYSTEM ENTERS DISCONNECTED STATE.';
	THIS^.pMachine^.SetState(THIS^.pMachine^.DisconnectedState);
END_IF
END_METHOD

METHOD PUBLIC PressDischarge
END_METHOD

METHOD PUBLIC Reset
END_METHOD

METHOD PUBLIC ResetContactors
VAR
	nIdx					: INT := 0; 
	bBypassContactors		: ARRAY[0..1] OF BOOL; 
	bMainContactors			: ARRAY[0..1] OF BOOL; 
END_VAR
FOR nIdx := 0 TO 1 BY 1 DO 
	bBypassContactors[nIdx] := FALSE;
	bMainContactors[nIdx] := FALSE; 
END_FOR

THIS^.pMachine^.BypassContactors := bBypassContactors; // Reset every contactor 
THIS^.pMachine^.MainContactors := bMainContactors;
END_METHOD

METHOD PUBLIC ResetTimer
THIS^.pMachine^.charge_TON.IN := FALSE;
END_METHOD

METHOD PUBLIC Stop
THIS^.pMachine^.SetState(THIS^.pMachine^.ErrorState);
END_METHOD

METHOD PUBLIC TimerDone
END_METHOD

END_FUNCTION_BLOCK

// ---- POUs/FB_ErrorState.TcPOU
FUNCTION_BLOCK INTERNAL FB_ErrorState IMPLEMENTS I_State
VAR
	pMachine 			: POINTER TO FB_MACHINE;
END_VAR

METHOD PUBLIC Check
THIS^.ResetContactors();
THIS^.ResetTimer();
END_METHOD

PROPERTY Description : STRING
GET
Description := 'ERROR';
END_GET
END_PROPERTY

METHOD PUBLIC FB_init
VAR_INPUT
	bInitRetains : BOOL; // if TRUE, the retain variables are initialized (warm start / cold start)
	bInCopyCode : BOOL;  // if TRUE, the instance afterwards gets moved into the copy code (online change)
	
	pMachine : POINTER TO FB_MACHINE;
END_VAR
THIS^.pMachine := pMachine;
END_METHOD

METHOD PUBLIC PressButton
END_METHOD

METHOD PUBLIC PressDischarge
END_METHOD

METHOD PUBLIC Reset
THIS^.pMachine^.SetState(THIS^.pMachine^.DisconnectedState);
END_METHOD

METHOD PUBLIC ResetContactors
VAR
	nIdx					: INT := 0; 
	bBypassContactors		: ARRAY[0..1] OF BOOL; 
	bMainContactors			: ARRAY[0..1] OF BOOL; 
END_VAR
FOR nIdx := 0 TO 1 BY 1 DO 
	bBypassContactors[nIdx] := FALSE;
	bMainContactors[nIdx] := FALSE; 
END_FOR

THIS^.pMachine^.BypassContactors := bBypassContactors; // Reset every contactor 
THIS^.pMachine^.MainContactors := bMainContactors;
END_METHOD

METHOD PUBLIC ResetTimer
THIS^.pMachine^.charge_TON.IN := FALSE;
END_METHOD

METHOD PUBLIC Stop
END_METHOD

METHOD PUBLIC TimerDone
END_METHOD

END_FUNCTION_BLOCK

// ---- POUs/FB_FileWriter.TcPOU
FUNCTION_BLOCK FB_FileWriter
VAR_INPUT
	sFilePath					: T_MaxString; 
	sFileName					: T_MaxString;
	sNetId						: STRING; // NetId of the target, leave empty for local
END_VAR
VAR CONSTANT
	nArrBufferSize				: INT := 1000; 	
END_VAR
VAR
    fbFileOpen  				: FB_FileOpen;
    fbFilePuts  				: FB_FilePuts;
    fbFileClose 				: FB_FileClose;
    nFileHandle 				: UINT;
	
    arrBuffer   				: ARRAY[0..nArrBufferSize] OF T_MaxString;
    eFileWriteState 			: (IDLE, OPEN_FILE, WRITE_TO_FILE, CLOSE_FILE, ERROR);
END_VAR

CASE eFileWriteState OF
    IDLE:
        // Make sure all the file writing FBs are ready for use (trigger on execute)
        Init();
        
        // We have pending data to be written
        IF arrBuffer[0] <> '' THEN // Makes sure that the first element of the array is not an empty string 
            eFileWriteState := OPEN_FILE;
        END_IF
        
    OPEN_FILE:
        // Opens a file for writing at the end of the file (append). 
        // If the file does not exist, a new file is created.
        fbFileOpen(
            bExecute    := TRUE,
            sNetId      := sNetId,
            sPathName   := CONCAT(sFilePath, sFileName),
            nMode       := FOPEN_MODEAPPEND);
            
        IF fbFileOpen.bError THEN
            eFileWriteState := ERROR;
        ELSIF NOT fbFileOpen.bBusy THEN
            nFileHandle := fbFileOpen.hFile;
            fbFileOpen(bExecute := FALSE);
            eFileWriteState := WRITE_TO_FILE;
        END_IF
    
    WRITE_TO_FILE:
        fbFilePuts(
            bExecute    := TRUE,
            sNetId      := sNetId,
            hFile       := nFileHandle,
            sLine       := arrBuffer[0]); // Write the first element of the buffer
        
        IF fbFilePuts.bError THEN
            eFileWriteState := ERROR;
        ELSIF NOT fbFilePuts.bBusy THEN
            fbFilePuts(bExecute := FALSE);
            RotateBuffer(); // Remove the written data from the buffer
            eFileWriteState := CLOSE_FILE;
        END_IF
    
    CLOSE_FILE:
        fbFileClose(
            bExecute := TRUE,
            sNetId      := sNetId,
            hFile       := nFileHandle);
            
        IF fbFileClose.bError THEN
            eFileWriteState := ERROR;
        ELSIF NOT fbFileClose.bBusy THEN
            nFileHandle := 0;
            eFileWriteState := IDLE;
        END_IF      
    
    ERROR:
        // Error, clear the handle and go back to idle
        nFileHandle := 0;
        eFileWriteState := IDLE;
END_CASE

PROPERTY PUBLIC FileWriteState : STRING
GET
CASE eFileWriteState OF
    IDLE: 
        FileWriteState := 'IDLE';
    OPEN_FILE: 
        FileWriteState := 'OPEN_FILE';
    WRITE_TO_FILE: 
        FileWriteState := 'WRITE_TO_FILE';
    CLOSE_FILE: 
        FileWriteState := 'CLOSE_FILE';
    ERROR: 
        FileWriteState := 'ERROR';
ELSE
    FileWriteState := 'UNKNOWN';
END_CASE
END_GET
END_PROPERTY

METHOD PRIVATE Init
fbFileClose(bExecute := FALSE);
fbFileOpen(bExecute := FALSE);
fbFilePuts(bExecute := FALSE);
END_METHOD

METHOD PRIVATE InsertToBuffer 
VAR_INPUT
	value					: STRING;
END_VAR
VAR
    nBufferIndex    : INT;
END_VAR
FOR nBufferIndex := 0 TO nArrBufferSize BY 1 DO
    IF arrBuffer[nBufferIndex] = '' THEN
        // We found the free spot in the buffer, insert the value to this place
        arrBuffer[nBufferIndex] := value;
        EXIT;
    END_IF
END_FOR
END_METHOD

METHOD PRIVATE RotateBuffer

VAR
    nIndex  : int := 0;
END_VAR
FOR nIndex := 0 TO nArrBufferSize - 1 BY 1 DO
    // We can exit when we reached the empty slot in the buffer
    IF arrBuffer[nIndex] = '' THEN
        EXIT;
    END_IF
    // FIFO, removing first element in the array copying the next, etc...
    arrBuffer[nIndex] := arrBuffer[nIndex+1];
END_FOR
arrBuffer[nArrBufferSize-1] := ''; // Clear the last element after rotation
END_METHOD

METHOD PUBLIC WriteToFile
VAR_INPUT
    message : T_MaxString;
END_VAR
InsertToBuffer(value := message);
END_METHOD

END_FUNCTION_BLOCK

// ---- GlobalTextList.TcGTLO
TEXTLIST GlobalTextList
  250 = '%d'
  613 = '%n'
  534 = '%s'
  442 = 'ACKNOWLEDGE'
  65 = 'BYPASS CONTACTORS :'
  386 = 'BYPASS CONTACTORS FB :'
  675 = 'CONTACTORS :'
  535 = 'CURRENT ID'
  718 = 'CURRENT ID :'
  597 = 'CURRENTS :'
  892 = 'DISCHARGE'
  328 = 'FILE WRITER STATE: '
  443 = 'FILE WRITER STATES : '
  615 = 'LOGS :'
  958 = 'MAIN CONTACTORS :'
  786 = 'MAIN CONTACTORS FB :'
  227 = 'MESSAGES :'
  52 = 'Start New Job'
  353 = 'STATE MACHINE STATE :'
  28 = 'VOLTAGES :'
END_TEXTLIST

// ---- VISUs/Visualisation.TcVIS
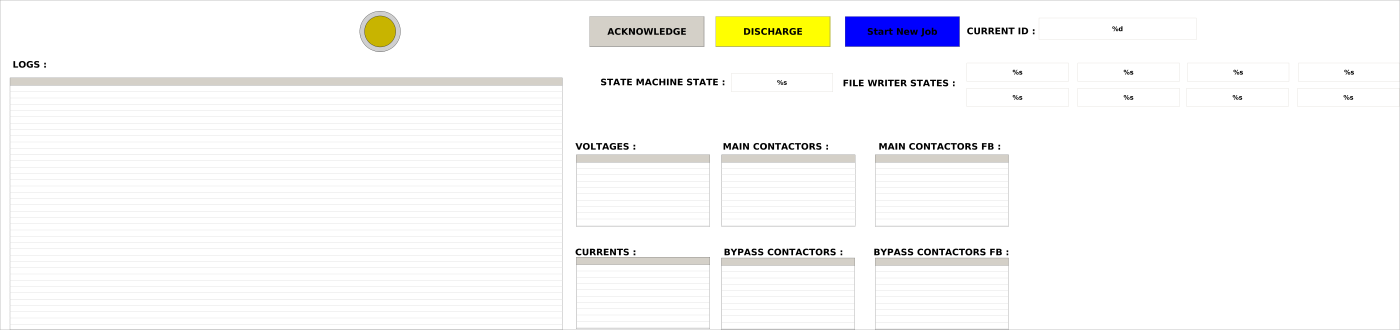
VISUALIZATION Visualisation  // 5552x1312
    Table (39,309 2191x1003), data array: MAIN.sLog
        p3854506369: MAIN.sLog[INDEX]
    Button (2338,65 455x121), "ACKNOWLEDGE", colour toggle: MAIN.b_user_button
        OnMouseDown: execute { MAIN.b_user_button := TRUE; }
        OnMouseUp: execute { MAIN.b_user_button := FALSE; }
    Textfield (2900,291 403x74), "%s", text variable: MAIN.sState
    Label (47,229 340x55), "LOGS :"
    Table (2285,615 530x285), data array: MAIN.n_V_sensors_scaled
        p3854506369: MAIN.n_V_sensors_scaled[INDEX]
    Table (2285,1022 530x285), data array: MAIN.n_A_sensors_scaled
        p3854506369: MAIN.n_A_sensors_scaled[INDEX]
    Label (2279,555 340x55), "VOLTAGES :"
    Label (2278,975 340x55), "CURRENTS :"
    Table (2861,615 530x285), data array: MAIN.b_main_contactors
        p3854506369: MAIN.b_main_contactors[INDEX]
    Label (2863,555 445x55), "MAIN CONTACTORS :"
    Label (2867,975 508x55), "BYPASS CONTACTORS :"
    Table (2860,1025 530x285), data array: MAIN.b_bypass_contactors
        p3854506369: MAIN.b_bypass_contactors[INDEX]
    Table (3470,615 530x285), data array: MAIN.b_main_contactors_fb
        p3854506369: MAIN.b_main_contactors_fb[INDEX]
    Label (3481,555 517x55), "MAIN CONTACTORS FB :"
    Label (3461,975 554x55), "BYPASS CONTACTORS FB :"
    Table (3470,1025 530x285), data array: MAIN.fbMachine.bBypassContactorsFB
        p3854506369: MAIN.fbMachine.bBypassContactorsFB[INDEX]
    Button (2838,65 455x121), "DISCHARGE", colour toggle: MAIN.b_discharge
        OnMouseDown: execute { MAIN.b_discharge :=TRUE; }
        OnMouseUp: execute { MAIN.b_discharge := FALSE; }
    Button (3351,65 455x121), "Start New Job", colour toggle: MAIN.bStartNewJob
        OnMouseDown: execute { MAIN.bStartNewJob := NOT(MAIN.bStartNewJob) }
        OnMouseUp: execute { MAIN.b_discharge := FALSE; }
    Textfield (3834,250 403x74), "%s", text variable: MAIN.s_FBStates[0]
    Textfield (3834,350 403x74), "%s", text variable: MAIN.s_FBStates[2]
    Textfield (4274,250 403x74), "%s", text variable: MAIN.s_FBStates[1]
    Textfield (4274,350 403x74), "%s", text variable: MAIN.s_FBStates[3]
    Label (2378,299 523x55), "STATE MACHINE STATE :"
    Label (3339,303 477x55), "FILE WRITER STATES :"
    Textfield (4120,71 624x87), "%d", text variable: MAIN.nIteration
    Label (3831,96 276x55), "CURRENT ID :"
    Lamp1 (1413,15 189x220), variable: MAIN.b_resetLed, style: Lamp-Lamp1-Yellow
    Textfield (4709,250 403x74), "%s", text variable: MAIN.s_FBStatesContactors[0]
    Textfield (4706,350 403x74), "%s", text variable: MAIN.s_FBStatesContactors[2]
    Textfield (5149,250 403x74), "%s", text variable: MAIN.s_FBStatesContactors[1]
    Textfield (5146,350 403x74), "%s", text variable: MAIN.s_FBStatesContactors[3]
END_VISUALIZATION
